(*======================================================================================================================================*)
(*FB_TasterBusSimple:	Einfache RS485 Kommunikation für Haus-bus.de Komponenten zum testen 	
						Achtung: Bei dem 6 Fach Taster ist zu Beachten, dass es nur 4 Externe EA/s gibt also 4 LEDs und 4 Taster *)
(*
Date          	| Version    	| created under        	| Author          	| Remark *)
(*====================================================================================================================================================*)
(*29/04/2025   	| 1.00      		| TC3		  		| N.Kersting       | first release *)
(*02/05/2025   	| 1.01      		| TC3		  		| N.Kersting       | Events für die Buttons werden erfolgreich verarbeitet *)
(*02/05/2025   	| 1.02      		| TC3		  		| N.Kersting       | Events für Temp, Helligkeit, Fuehctigkeit erfolgreich Implementier *)
(*02/05/2025   	| 1.03      		| TC3		  		| N.Kersting       | Set Schrittkette für Reset und LED Helligkeit erfolgreich Implementier*)
(*02/05/2025   	| 1.04      		| TC3		  		| N.Kersting       | In und Out Strukturen Implementiert und Startup nach Reset *)
(*02/05/2025   	| 1.05      		| TC3		  		| N.Kersting       | Pingabgfrage*)
(*02/05/2025   	| 1.06      		| TC3		  		| N.Kersting       | Reset Startup Implementiert*)
(*03/05/2025   	| 1.07      		| TC3		  		| N.Kersting       | Ping wird nun bei PLC Reset auch gestaret und Execute wird richtig verwendet*)
(*04/05/2025   	| 1.08      		| TC3		  		| N.Kersting       | Hintergrundbeleuchtung und Zähler für die Tatser Implementiert *)
(*04/05/2025   	| 1.09      		| TC3		  		| N.Kersting       | Neuen Baustein zum Einheitlichen versenden von Telegrammen Implementiert *)
(*05/05/2025   	| 2.00      		| TC3		  		| N.Kersting       | Komplett neuen Baustein, mit Externer Receive Auswertung und neuem Ping Baustein *)
(*06/05/2025   	| 2.01      		| TC3		  		| N.Kersting       | Externe LEDs Implementiert *)
(*07/05/2025   	| 2.02      		| TC3		  		| N.Kersting       | Im Startup wird nun auf die Device ID geachtet *)
(*08/05/2025   	| 2.03      		| TC3		  		| N.Kersting       | Externe LEDs sind nun Umschaltbar/ LEDs oder normaler Ausgang (Betriefft die Hintergrundbeleuchtung) -> Weniger Busauslastung *)
(*09/05/2025   	| 2.04      		| TC3		  		| N.Kersting       | Ping Versuche Implementiert mit Globalen Parametern *)
(*09/05/2025   	| 2.05      		| TC3		  		| N.Kersting       | Ping für Taster nun Auch automatisch durch Empfang von sämtlichen Telegrammen*)
(*09/05/2025   	| 2.06      		| TC3		  		| N.Kersting       | Bugfix im Startup Angepasst! nur noch Hintergrundbeleuchtung setzen! *)
(*10/05/2025   	| 3.00      		| TC3		  		| N.Kersting       | Umstellung auf Externe FiFo Sendebaustein *)
(*13/05/2025   	| 3.01      		| TC3		  		| N.Kersting       | Viele Bugs gefixt, bei Änderung der Ausgängen wird nun eine Anforderung gesetzt  *)
(*13/05/2025   	| 3.02      		| TC3		  		| N.Kersting       | Test für Github *)
(*22/05/2025   	| 3.03      		| TC3		  		| N.Kersting       | Grundaufbau vom BusTaster, jetzt allerdings für ein CYD mit den gleichen Funktionen *)
(*22/05/2025   	| 3.04      		| TC3		  		| N.Kersting       | ServiceFunktionen für CYD Hinzugefügt (Wifi und Webserver Starten)*)
(*23/05/2025   	| 3.05      		| TC3		  		| N.Kersting       | Neue eigene Input Struktur für das CYD Implementiert*)
(*23/05/2025   	| 3.06      		| TC3		  		| N.Kersting       | Auto - Input Fault Detection implementiert (Wenn Taster zu lange aktiviert bleibt ) *)
(*26/05/2025   	| 3.07      		| TC3		  		| N.Kersting       | Updaten im Com Check Baustein, der Zyklische Ping vom CYD wird nun erkannt ) *)
(*28/05/2025   	| 3.08      		| TC3		  		| N.Kersting       | Neuen Einfachen Ping Baustein, welcher nicht sendet, nur auswertet implementiert *)
(*====================================================================================================================================================*)
FUNCTION_BLOCK fb_CYDBus6F
VAR_INPUT
	I_FifoID			:INT;
	I_bPingStart		:BOOL;						(* Ping Done vom Vorheriegen*)
	I_stInput			:ST_BusCYD6F_Input;
	I_StringReceived	:STRING(255);
END_VAR
VAR_OUTPUT
	Q_sFiFoSend			:STRING(255);
   	Q_stOutput			:ST_BusTaster6F_Output;
	Q_stCnt				:ST_BusTaster6F_Cnt;
END_VAR
VAR
(*----------------------------------------------*)
(* Interne Parameter*)
(*----------------------------------------------*)		
	bSetExecute			:BOOL := TRUE;				(* Aktiviert die Schrittketten, welche Telegramme versenden *)
	bCheckPing			:BOOL := TRUE;				(* Ping Checken Schrittkette Aktivieren *)
	sStartZeichen		:BYTE := 16#FD;				(* Startzeichen Präfix *)
	sEndZeichen			:BYTE := 16#FE;				(* Endzeichen Suffix *)
	iAnzResetSend		:INT := 2;					(* Anzahl der Sendeversuche bei Reset *)
	tPingTimer			:TIME:= T#5S;				(* Zeit, bis wiederholend der Ping versendet wird *)
	tReceiveTimeout		:TIME:= T#2S;				(* Zeit, bis die Event Schrittkette für das Empfangen Automatisch neu Startet*)
	tStartupLEDOn		:TIME:= T#4S;				(* Zeit, wie Lange die LEDS beim Startup kurz eingeschaltet werden *)
	tResetTimeout		:TIME:= T#25S;				(* Zeit, bis bei einem Reset es zu einem Fehler kommt, wenn kein Ping empfangen wird *)
	tResetReboot		:TIME:= T#10S;				(* Zeit, die nach einem Reset Abgewaretet wird damit das Gerät neustarten kann*)
	tResetStartup		:TIME:= T#5S;				(* Zeit, die nach einem Reset Abgewaretet wird bis ein Startup ausgeführt wird nach dem erhalt des Pings vom Gerät*)
	tStartupAfterReset	:TIME := T#5S;				(* Zeit, wann das Startup Zurückgesetzt wird, wenn der Ping verloren wird *)
	bInputFaultDetect	:BOOL := TRUE;				(* Prüft die Eingänge ob sie zu lange geschaltet wurden und führt ein reset des eingangs aus *)
	tInputFaultDetect	:TIME := T#10S;				(* Prüft die Eingänge ob sie zu lange geschaltet wurden und führt ein reset des eingangs aus *)
(*----------------------------------------------*)
(*	Service Funktionen Aktivieren *)
(*----------------------------------------------*)	
	bWebServer			:BOOL := FALSE;				(* zuerst funktion auswählen (bWebserver/ bWifi, bService) und dann mit bStartServiceMode ausführen *)
	bWifi				:BOOL := FALSE;				(* zuerst funktion auswählen (bWebserver/ bWifi, bService) und dann mit bStartServiceMode ausführen *)
	bService			:BOOL := FALSE;				(* zuerst funktion auswählen (bWebserver/ bWifi, bService) und dann mit bStartServiceMode ausführen *)
	(*	*)
	bStartServiceMode	:BOOL := FALSE;				(* zuerst ServiceMode Aktivieren und dann mit bStartServiceMode ausführen *)
	
	(* Speichern der zustände *)
	bMemWebServer		:BOOL;
	bMemWifi			:BOOL;
	bMemService			:BOOL;
	
(*----------------------------------------------*)
(* Strings *)
(*----------------------------------------------*)			
	sSendString			:STRING(255);
	sFiFoSend			:STRING(255);
	sReceived			:STRING(255);
	sLastSendString		:STRING(255);
	sStateReset			:STRING;
(*----------------------------------------------*)
(* Funktionsbausteine *)
(*----------------------------------------------*)
	fbBusTasterEvent	:ARRAY[1..6] OF fb_BusTasterEvent;		(* Interne 6 Taster Abfragen *)
	fbBusTasterEventExt	:ARRAY[1..6] OF fb_BusTasterEvent;		(* Externe 6 Eingänge Abfragen *)
	fbBusTempEvent		:fb_BusTempEvent;
	fbBusBrsEvent		:fb_BusBrsEvent;
	fbBusRhdEvent		:fb_BusRhdEvent;
	fbStringConvTB6F	:fb_StringConvTB6F;
	fbStringConvWeb		:fb_StringConvCYDWeb;
	fbStringConvWifi	:fb_StringConvCYDWifi;
	fbStringConvService	:fb_StringConvCYDService;
	fbPing				:fb_RS485Ping;
(*----------------------------------------------*)
(* Indexe *)
(*----------------------------------------------*)	
	iDeviceStartup		:INT :=0;	(* Startup Schrittkette *)
	sDeviceStartup		:STRING;
    iState     			:INT := 0;
	iStepSet			:INT;
	i,h,j,l,e			:INT;
	idxLED				:INT;
	idxBtn				:INT := 1;
	
	iDimmMem			:ARRAY[1..6] OF INT;
	iDimmMemExt			:ARRAY[1..6] OF INT;
	iDimmBGAnf			:INT;
	iDimmAnf			:ARRAY[1..6] OF INT;
	iDimmAnfExt			:ARRAY[1..6] OF INT;
	
	iDimmBgMem			:INT;
	cntChangesDimm		:INT;
	cntChangesDimmExt	:INT;
	icntResetSend		:INT;
	iMaxPingTry			:INT := 5;
(*----------------------------------------------*)
(* Timer/Trigger *)
(*----------------------------------------------*)		
	r_trigStartupAfterReset	:r_trig;
	r_TrigReset				:r_trig;		
	r_TrigCountBtn			:ARRAY[1..6] OF r_trig;
	
	tonStartupAfterReset	:ton;
	tonReceiveTimeout		:ton;
	tonResetTimeout			:ton;
	tonResetDone			:ton;
	tonStepStartup			:ton;
(*----------------------------------------------*)
(* Status *)
(*----------------------------------------------*)			
	bPingOK					:BOOL;
	bErrorEvent				:BOOL;
	bErrorPing				:BOOL;
	bErrorSet				:BOOL;
	bErrorReset				:BOOL;
	bResetBusy				:BOOL;
	bResetDone				:BOOL;
	bResetAutoStart			:BOOL;
	bStartupStart			:BOOL;
	bStartupDone			:BOOL;	
	bMemExt					:BOOL;
	bStartUpCheckPing		:BOOL;
	bActivateSend			:BOOL;
	bReadyToPing			:BOOL;
	bSendeAnforderung		:BOOL;
	bSendeAnforderungExt	:BOOL;
	bSendeAnforderungBG		:BOOL;
	
END_VAR

(*============================================================================================*)
(* Parameter *)
tPingTimer :=		GVL_HausBus_Parameter.cTimePingTimeCYD;
tReceiveTimeout :=	GVL_HausBus_Parameter.cTimeReceiveTimeoutCYD;
bCheckPing :=		GVL_HausBus_Parameter.bUseCYDPing;
iMaxPingTry :=		GVL_HausBus_Parameter.cMaxPingTry;

(* Service *)
bWebServer :=			I_stInput.bWebServer;
bWifi :=				I_stInput.bWifi;
bService :=				I_stInput.bService;
bStartServiceMode :=	I_stInput.bServiceMode;

(*============================================================================================*)
(* Startup Zurücksetzen Reset *)
r_TrigReset(CLK := I_stInput.bReset);

(* Startup Zurücksetzen bei Busverlust *)
tonStartupAfterReset(
	IN := NOT bPingOK
			AND bCheckPing,
	PT:= tStartupAfterReset);

r_trigStartupAfterReset
	(CLK := tonStartupAfterReset.Q);
	
IF NOT I_stInput.bExecute
	OR r_TrigReset.Q
	OR r_trigStartupAfterReset.Q
THEN
	iDeviceStartup := 0;
ELSIF
	bStartServiceMode
THEN	
	iDeviceStartup := 5;
END_IF

(*============================================================================================*)
(* Ping Dauerhaft Senden*)
ac02_Ping();
	
(*============================================================================================*)
(* Startup Schrittkette *)
CASE iDeviceStartup OF
(*============================================================================================*)
0: 	sDeviceStartup := 'INIT';
	bResetDone := FALSE;
	bStartupDone := FALSE;
	bStartupStart := FALSE;
	bResetAutoStart := FALSE;
	bStartUpCheckPing := FALSE;
	bActivateSend := FALSE;
	bReadyToPing := TRUE;
	bMemWebServer :=FALSE;
	bMemWifi :=	FALSE;
	bMemService	:= FALSE;
	
	sFiFoSend := ''; 
	iStepSet := 0;
	
	IF 	I_stInput.bExecute
	THEN
		iDeviceStartup := iDeviceStartup+1;
	END_IF
(*============================================================================================*)
1: 	sDeviceStartup := 'Device ID Prüfen';
	
	IF  I_stInput.diID <> 0
	THEN
		iDeviceStartup := iDeviceStartup+1;
	ELSE
		sDeviceStartup := 'ERROR- Device ID Prüfen';
	END_IF
(*============================================================================================*)
2: 	sDeviceStartup := 'Verbindung Prüfen';
	bActivateSend := TRUE;	(* Senden Aktivieren *)
	iDeviceStartup := iDeviceStartup+1;
	
	(*
	sDeviceStartup := CONCAT(sDeviceStartup,fbRS485ComCheck.Q_sState);
	
	IF fbRS485ComCheck.Q_bComOk
		OR NOT bCheckPing
	THEN
	END_IF*)

(*============================================================================================*)
3: 	sDeviceStartup := 'Reset Ausführen';	
	bActivateSend := TRUE;	(* Senden Aktivieren *)
	
	(*	RESET Device *)
	ac01_SetReset();
	bResetAutoStart := TRUE;
	
	sDeviceStartup :=	CONCAT(sDeviceStartup,sStateReset);
	
	IF bResetDone
	THEN
		iStepSet := 0;
		iDeviceStartup := iDeviceStartup+1;
	END_IF

(*============================================================================================*)
4: 	sDeviceStartup := 'Startup Ausführen';
		
	(* LED Setzen *)
	ac01_SetLED();
	
	bStartupStart := TRUE;
	
	IF bStartupDone 
	THEN
		bStartupStart := FALSE;
		iDeviceStartup := 999;
	END_IF

(*============================================================================================*)
5:	sDeviceStartup := 'Service Funktionen Steuern';
	ac01_SetService();

	IF NOT bStartServiceMode 
	THEN
		iStepSet := 0;
		iDeviceStartup := 0;
	END_IF
	
(*============================================================================================*)
999: 
	(*bReadyToPing := NOT fbRS485SendCmd.Q_bBusy;*)
	
	(* LED Setzen *)
	ac01_SetLED();
	
	(* Events Auslesen *)
	ac00_Event();
	
	(* Zähler *)
	ac10_Counter();
	
	sDeviceStartup := 'Startup Ausgeführt- Gerät im OP';
	
END_CASE

(*============================================================================================*)
(* Sendebaustein *)
IF bActivateSend
THEN
	Q_sFiFoSend :=	sFiFoSend;
END_IF

(*============================================================================================*)	
(* Zähler *)
ac10_Counter();
	
(*============================================================================================*)
(* Outputs *)
Q_stOutput.bCOM :=		bPingOK;

Q_stOutput.bError := 	bErrorEvent
						OR bErrorPing
						OR bErrorSet
						OR (NOT bPingOK
						AND bCheckPing);
						
Q_stOutput.bStartupDone	:=	bStartupDone;

Q_stOutput.sState :=	CONCAT(I_stInput.sName,'| ');
Q_stOutput.sState :=	CONCAT(Q_stOutput.sState, sDeviceStartup);

ACTION ac00_Event:
(*============================================================================================*)
(*	EVENT Schrittkette *)
(*============================================================================================*)
sReceived := I_StringReceived;
	
FOR i := 1 TO 6 BY 1 DO 
	fbBusTasterEvent[i](
		I_bFaultDetection	:=	bInputFaultDetect,
		I_tFaultDetectTime	:=	tInputFaultDetect,
		I_sID:= 				DINT_TO_STRING(I_stInput.diID), 
		I_sInstID:= 			INT_TO_STRING(i+16), 
		I_sReceivedString:= 	sReceived, 
		Q_bOut=> 				Q_stOutput.bButtons[i]);
	
	fbBusTasterEventExt[i](
		I_sID:= 				DINT_TO_STRING(I_stInput.diID), 
		I_sInstID:= 			INT_TO_STRING(i+32), 
		I_sReceivedString:= 	sReceived, 
		Q_bOut=> 				Q_stOutput.bButtonsExt[i]);
		
	fbBusTempEvent(
		I_sID:= 				DINT_TO_STRING(I_stInput.diID), 
		I_sInstID:= 			'1', 
		I_sReceivedString:= 	sReceived, 
		Q_lrTemp=> 				Q_stOutput.lrTemp);
		
	fbBusBrsEvent(
		I_sID:= 				DINT_TO_STRING(I_stInput.diID), 
		I_sInstID:= 			'1', 
		I_sReceivedString:= 	sReceived, 
		Q_lrBrs=> 				Q_stOutput.lrBrs);
		
	fbBusRhdEvent(
		I_sID:= 				DINT_TO_STRING(I_stInput.diID), 
		I_sInstID:= 			'1', 
		I_sReceivedString:= 	sReceived, 
		Q_lrRhd=> 				Q_stOutput.lrRhd);
END_FOR
END_ACTION

ACTION ac01_SetLED:
(*============================================================================================*)
(*	LED Helligkeit Setzen/ Startup Schrittkette *)
(*============================================================================================*)

(* Einfaches Setzen der LED Helligkeiten (0-100 Prozent *)
(* Neu, es werden alle LEDs zu einem String zusammengefügt und Gleichzeitig gesetzt *)
tonStepStartup(
	PT:= tStartupLEDOn);
	
cntchangesDimm := 0;
cntChangesDimmExt :=0;
	
FOR l := 1 TO 6 BY 1 DO
	IF iDimmMem[l] <> I_stInput.iLED[l]
	THEN
		cntChangesDimm := cntChangesDimm +1;
	END_IF

	IF  iDimmMemExt[l]<> I_stInput.iLEDExt[l]
	THEN
		cntChangesDimmExt := cntChangesDimmExt +1;
	END_IF
END_FOR

CASE iStepSet OF
(*============================================================================================*)
0:	(* INIT und warten auf Change *)				
	tonStepStartup.IN := FALSE;
	sFiFoSend := ''; 
	
	(* Änderungs- Anforderungen Prüfen*)
	FOR e := 1 TO 6 BY 1 DO
		IF cntChangesDimm<>0
		THEN
			(* Helligkeitanforderung Interne LEDs speichern *)
			bSendeAnforderung := TRUE;
			iDimmAnf[e] 	:= I_stInput.iLED[e];
		END_IF
		
		IF cntChangesDimmExt <> 0
		THEN
			(* Helligkeitanforderung Externe LEDs speichern *)
			bSendeAnforderungExt := TRUE;
			iDimmAnfExt[e] 	:= I_stInput.iLEDExt[e];
		END_IF
		
		IF I_stInput.iLEDBg <>iDimmBgMem
		THEN
			(* Helligkeitsanforderung Hintergrundbeleuchtung *)
			bSendeAnforderungBG := TRUE;
			iDimmBGAnf		:= I_stInput.iLEDBg;
		END_IF
	END_FOR
	
	(* Reagieren auf Anforderungen *)
	IF ((bSendeAnforderung
		OR bSendeAnforderungExt
		OR bSendeAnforderungBG)
		AND bSetExecute)
		AND NOT bStartupStart
	THEN
		(* Helligkeitsvorgaben speichern in Mem Arrays *)
		FOR h := 1 TO 6 BY 1 DO
			iDimmMem[h] := I_stInput.iLED[h];
			iDimmMemExt[h] := I_stInput.iLEDExt[h];
			iDimmBgMem := I_stInput.iLEDBg;
		END_FOR
		
		iStepSet := 10;
	ELSIF
		bStartupStart
	THEN
		iStepSet := 100;	(* Startup *)
	END_IF
	
(*============================================================================================*)
10:	(* Prüfen welche Anforderung ausgeführt werden soll *)	
	IF	bSendeAnforderungBG
		AND NOT bSendeAnforderung
		AND NOT bSendeAnforderungExt 
	THEN
		iStepSet := 22;(* Direkt nur die Hintergrund Helligkeit setzen *)
	ELSE
		(* Nur Interne LEDs Schreiben *)
		IF bSendeAnforderung
			AND NOT bSendeAnforderungExt
			AND NOT bSendeAnforderungBG
		THEN
			fbStringConvTB6F(
				I_bSetBackground :=	FALSE,
				I_bReset :=			FALSE,
				I_bExtLED :=		FALSE,
				I_bHasExtLED :=		I_stInput.bExtOutLED,
				I_diID:= 			I_stInput.diID, 
				I_iLED:= 			iDimmAnf, 
				I_iLEDExt:=			iDimmAnfExt,
				I_iLEDBg:= 			iDimmBGAnf,		 
				I_sStartZeichen:= 	sStartZeichen, 
				I_sEndZeichen:= 	sEndZeichen, 
				Q_sConvString=> 	sSendString);
				
			(* Senden an FiFo*)
			IF GVL_RS485FiFoSend.bSendDoneFiFo[I_FifoID]
			THEN
				sFiFoSend :=	sSendString;
			END_IF
			IF NOT GVL_RS485FiFoSend.bSendDoneFiFo[I_FifoID]
			THEN
				bSendeAnforderung := FALSE;
				sLastSendString :=	sFiFoSend;
				iStepSet := 20;
			END_IF
		ELSIF
			(* Nur Externe LEDs Schreiben *)	
			bSendeAnforderungExt
			AND NOT bSendeAnforderung
			AND NOT bSendeAnforderungBG
		THEN
			fbStringConvTB6F(
				I_bSetBackground :=	FALSE,
				I_bReset :=			FALSE,
				I_bExtLED :=		TRUE,
				I_bHasExtLED :=		I_stInput.bExtOutLED,
				I_diID:= 			I_stInput.diID, 
				I_iLED:= 			iDimmAnf, 
				I_iLEDExt:=			iDimmAnfExt,
				I_iLEDBg:= 			iDimmBGAnf,				 
				I_sStartZeichen:= 	sStartZeichen, 
				I_sEndZeichen:= 	sEndZeichen, 
				Q_sConvString=> 	sSendString);
			
			(* Senden an FiFo*)
			IF GVL_RS485FiFoSend.bSendDoneFiFo[I_FifoID]
			THEN
				sFiFoSend :=	sSendString;
			END_IF
			IF NOT GVL_RS485FiFoSend.bSendDoneFiFo[I_FifoID]
			THEN
				bSendeAnforderungExt := FALSE;
				sLastSendString :=	sFiFoSend;
				iStepSet := 20;
			END_IF
		ELSE
			(* Externe und Interne LEDs Schreiben *)
			bMemExt := TRUE; (* Speichern, damit anschließend noch die Externen LEDs gesetzt werden *)
			
			fbStringConvTB6F(
				I_bSetBackground :=	FALSE,
				I_bReset :=			FALSE,
				I_bExtLED :=		FALSE,
				I_bHasExtLED :=		I_stInput.bExtOutLED,
				I_diID:= 			I_stInput.diID, 
				I_iLED:= 			iDimmAnf, 
				I_iLEDExt:=			iDimmAnfExt,
				I_iLEDBg:= 			iDimmBGAnf,			 
				I_sStartZeichen:= 	sStartZeichen, 
				I_sEndZeichen:= 	sEndZeichen, 
				Q_sConvString=> 	sSendString);
			
			(* Senden an FiFo*)
			IF GVL_RS485FiFoSend.bSendDoneFiFo[I_FifoID]
			THEN
				sFiFoSend :=	sSendString;
			END_IF
			IF NOT GVL_RS485FiFoSend.bSendDoneFiFo[I_FifoID]
			THEN
				bSendeAnforderung := FALSE;
				bSendeAnforderungExt := FALSE;
				sLastSendString :=	sFiFoSend;
				iStepSet := 20;
			END_IF
		END_IF
	END_IF
(*============================================================================================*)	
20:	(* Warten bis nicht Busy *)	
	
	IF GVL_RS485FiFoSend.bSendDoneFiFo[I_FifoID]
	THEN
		sFiFoSend := ''; 
		IF NOT bMemExt
		THEN
			IF bSendeAnforderungBG
			THEN
				iStepSet := 22;
			ELSE
				iStepSet := 0;
			END_IF
		ELSE
			iStepSet :=	21;
		END_IF
	END_IF
	
(*============================================================================================*)	
21:	(* Externe LEDs Senden *)	
	bMemExt := FALSE;
	bSendeAnforderungExt := FALSE;
	
	fbStringConvTB6F(
		I_bSetBackground :=	FALSE,
		I_bReset :=			FALSE,
		I_bExtLED :=		TRUE,
		I_bHasExtLED :=		I_stInput.bExtOutLED,
		I_diID:= 			I_stInput.diID, 
		I_iLED:= 			iDimmAnf, 
		I_iLEDExt:=			iDimmAnfExt,
		I_iLEDBg:= 			iDimmBGAnf,				 
		I_sStartZeichen:= 	sStartZeichen, 
		I_sEndZeichen:= 	sEndZeichen, 
		Q_sConvString=> 	sSendString);
		
	(* Senden an FiFo*)
	IF GVL_RS485FiFoSend.bSendDoneFiFo[I_FifoID]
	THEN
		sFiFoSend :=	sSendString;
	END_IF
	IF NOT GVL_RS485FiFoSend.bSendDoneFiFo[I_FifoID]
	THEN
		sLastSendString :=	sFiFoSend;
		iStepSet := 20;
	END_IF
	
(*============================================================================================*)	
22:	(* Hintergrundbeleuchtung senden *)		
	bSendeAnforderungBG := FALSE;
	
	fbStringConvTB6F(
		I_bSetBackground :=	TRUE,
		I_bReset :=			FALSE,
		I_bExtLED :=		FALSE,
		I_bHasExtLED :=		I_stInput.bExtOutLED,
		I_diID:= 			I_stInput.diID, 
		I_iLED:= 			iDimmAnf, 
		I_iLEDExt:=			iDimmAnfExt,
		I_iLEDBg:= 			iDimmBGAnf,			 
		I_sStartZeichen:= 	sStartZeichen, 
		I_sEndZeichen:= 	sEndZeichen, 
		Q_sConvString=> 	sSendString);
		
	(* Senden an FiFo*)
	IF GVL_RS485FiFoSend.bSendDoneFiFo[I_FifoID]
	THEN
		sFiFoSend :=	sSendString;
	END_IF
	IF NOT GVL_RS485FiFoSend.bSendDoneFiFo[I_FifoID]
	THEN
		sLastSendString :=	sFiFoSend;
		iStepSet := 20;
	END_IF

(*============================================================================================*)	
(* Startup LEDS einmal Einschalten *)
100:	tonStepStartup.IN := TRUE;
	
	IF tonStepStartup.Q
	THEN
		iStepSet := 110;
	END_IF
	
(*============================================================================================*)
110:	(* String senden *)	
	tonStepStartup.IN := FALSE;
	
	fbStringConvTB6F(
		I_bSetBackground :=	TRUE,
		I_bExtLED :=		FALSE,
		I_bReset :=			FALSE,
		I_bHasExtLED :=		I_stInput.bExtOutLED,
		I_diID:= 			I_stInput.diID, 
		I_iLEDBg:= 			5,		 
		I_sStartZeichen:= 	sStartZeichen, 
		I_sEndZeichen:= 	sEndZeichen, 
		Q_sConvString=> 	sSendString);
			
	(* Senden an FiFo*)
	IF GVL_RS485FiFoSend.bSendDoneFiFo[I_FifoID]
	THEN
		sFiFoSend :=	sSendString;
	END_IF
	IF NOT GVL_RS485FiFoSend.bSendDoneFiFo[I_FifoID]
	THEN
		
		iStepSet := 111;
	END_IF
	
(*============================================================================================*)	
111:(* Warten bis nicht Busy *)	
	IF GVL_RS485FiFoSend.bSendDoneFiFo[I_FifoID]
	THEN
		sFiFoSend := ''; 
		tonStepStartup.IN := TRUE;
		
		IF tonStepStartup.Q
		THEN
			tonStepStartup.IN := FALSE;
			iStepSet := 120;
		END_IF
	END_IF
	
(*============================================================================================*)
120:	(* String senden *)	
	fbStringConvTB6F(
		I_bSetBackground :=	TRUE,
		I_bExtLED :=		FALSE,
		I_bReset :=			FALSE,
		I_bHasExtLED :=		I_stInput.bExtOutLED,
		I_diID:= 			I_stInput.diID, 
		I_iLEDBg:= 			100,		 
		I_sStartZeichen:= 	sStartZeichen, 
		I_sEndZeichen:= 	sEndZeichen, 
		Q_sConvString=> 	sSendString);
			
	(* Senden an FiFo*)
	IF GVL_RS485FiFoSend.bSendDoneFiFo[I_FifoID]
	THEN
		sFiFoSend :=	sSendString;
	END_IF
	IF NOT GVL_RS485FiFoSend.bSendDoneFiFo[I_FifoID]
	THEN
		iStepSet := 130;
	END_IF
	
(*============================================================================================*)	
130:(* Warten bis nicht Busy *)	
	IF GVL_RS485FiFoSend.bSendDoneFiFo[I_FifoID]
	THEN
		sFiFoSend := ''; 
			
		tonStepStartup.IN := TRUE;
	
		IF tonStepStartup.Q
		THEN
			bStartupDone := TRUE;
			tonStepStartup.IN := FALSE;
			bStartupStart := FALSE;
			iStepSet := 10;	(* Anschließend noch einmal die Eingangs Helligkeit setzen *)
		END_IF
	END_IF	

END_CASE

(*bErrorSet := fbRS485SendCmd.Q_bError;*)
END_ACTION

ACTION ac01_SetReset:
(*============================================================================================*)
(*	RESET Schrittkette *)
(*============================================================================================*)
tonResetTimeout(
	PT := tResetTimeout);

tonResetDone();

(* Einfaches Setzen der LED Helligkeiten (0-100 Prozent *)
CASE iStepSet OF
(*============================================================================================*)
0:	sStateReset := 'INIT';
	
	IF (bSetExecute
		AND (I_stInput.bReset
		OR bResetAutoStart))
	THEN
		sFiFoSend := ''; 
		bStartupDone := FALSE;
		bResetDone := FALSE;
		tonResetTimeout.IN := FALSE;
		tonResetDone.IN := FALSE;
		icntResetSend := 0;
		
		(* Ausgänge alle auf 0 setzen *)
		FOR h := 1 TO 6 BY 1 DO
			fbBusTasterEvent[i](
				I_sReceivedString :='');
				
			fbBusTasterEventExt[i](
				I_sReceivedString :='');	
				
			iDimmMem[h] := 0;
			Q_stOutput.bButtons[h] := FALSE;
			Q_stOutput.lrTemp := 0;
			Q_stOutput.lrBrs := 0;
			Q_stOutput.lrRhd := 0;
		END_FOR
		
		fbBusTempEvent(
			I_sReceivedString :='',	
			I_bReset := TRUE);
			
		fbBusBrsEvent(
			I_sReceivedString :='',	
			I_bReset := TRUE);
			
		fbBusRhdEvent(
			I_sReceivedString :='',	
			I_bReset := TRUE);
		
		bPingOK := FALSE;
		
		iStepSet := iStepSet +1;
	END_IF

(*============================================================================================*)	
1:	sStateReset := 'Sende Reset Befehl';
	bResetBusy := TRUE;
	bErrorReset := FALSE;
	
	fbStringConvTB6F(
		I_bReset :=			TRUE,
		I_diID:= 			I_stInput.diID, 		 
		I_sStartZeichen:= 	sStartZeichen, 
		I_sEndZeichen:= 	sEndZeichen, 
		Q_sConvString=> 	sSendString);

	(* Senden an FiFo*)
	IF GVL_RS485FiFoSend.bSendDoneFiFo[I_FifoID]
	THEN
		sFiFoSend :=	sSendString;
	END_IF
	IF NOT GVL_RS485FiFoSend.bSendDoneFiFo[I_FifoID]
	THEN
		iStepSet := iStepSet+1;
	END_IF

(*============================================================================================*)
2:	sStateReset := 'Sende Reset Befehl';

	IF GVL_RS485FiFoSend.bSendDoneFiFo[I_FifoID]
	THEN
		sFiFoSend := ''; 
		fbStringConvTB6F(
			I_bReset :=			FALSE);
		iStepSet := 3;
				
	END_IF
	
(*============================================================================================*)	
3:	sStateReset := 'Reset durchgeführt, Warte auf Ping';
	tonResetDone.IN := TRUE;
	tonResetDone.PT := tResetReboot;
	
	fbBusTempEvent(I_bReset := FALSE);
	fbBusBrsEvent(I_bReset := FALSE);
	fbBusRhdEvent(I_bReset := FALSE);
	
	iState := 0;
	
	IF tonResetDone.Q
	THEN
		tonResetDone.IN := FALSE;
		iStepSet := 4;
	END_IF
	
(*============================================================================================*)	
4:	sStateReset := 'Warte auf Ping vom Gerät';	
	tonResetTimeout.IN := TRUE;
	bStartUpCheckPing := TRUE;
	
	IF bPingOK 
	(*	OR NOT bCheckPing*)
	THEN
		bErrorReset := FALSE;
		tonResetTimeout.IN := FALSE;
		iStepSet := 5;
	ELSIF
		tonResetTimeout.Q
	THEN
		sStateReset := 'Ping Timeout, keine Kommunikation';
		bErrorReset := TRUE;

		IF I_stInput.bReset
		THEN
			bResetBusy := FALSE;
			iStepSet := 0;
		END_IF
	END_IF

(*============================================================================================*)
5:	sStateReset := 'Startup Aktiv';
	
	tonResetDone.IN := NOT I_stInput.bReset;
	tonResetDone.PT := tResetStartup;
	sFiFoSend := ''; 
	
	IF tonResetDone.Q
	THEN
		fbStringConvTB6F(
			I_bReset :=			FALSE);
			
		sStateReset := 'Ping erhalten, Reset Erfolgreich';
		bResetAutoStart := FALSE;
		bResetDone := TRUE;
		bResetBusy := FALSE;
		iState := 0;
		iStepSet := 0;
	END_IF
END_CASE
END_ACTION

ACTION ac01_SetService:
(*============================================================================================*)
(*	RESET Schrittkette *)
(*============================================================================================*)
tonResetTimeout(
	PT := tResetTimeout);

tonResetDone();

(* Einfaches Setzen der LED Helligkeiten (0-100 Prozent *)
CASE iStepSet OF
(*============================================================================================*)
0:	sStateReset := 'INIT';
	
	IF bSetExecute
		AND (bMemWebServer <> bWebServer
		OR bMemWifi <> bWifi
		OR bMemService <> bService )
	THEN
		bMemWebServer :=	bWebServer;
		bMemWifi :=			bWifi;
		bMemService	:=		bService;
		
		sFiFoSend := ''; 
		tonResetTimeout.IN := FALSE;
		tonResetDone.IN := FALSE;
		icntResetSend := 0;
		
		iStepSet := iStepSet +1;
	END_IF

(*============================================================================================*)	
1:	sStateReset := 'Sende Webserver Befehl';
	fbStringConvWeb(
		I_diID:= 			I_stInput.diID,
		I_bWebOn:= 			bWebServer, 
		I_sStartZeichen:= 	sStartZeichen, 
		I_sEndZeichen:= 	sEndZeichen, 
		Q_sConvString=> 	sSendString);
	
	(* Senden an FiFo*)
	IF GVL_RS485FiFoSend.bSendDoneFiFo[I_FifoID]
	THEN
		sFiFoSend :=	sSendString;
	END_IF
	IF NOT GVL_RS485FiFoSend.bSendDoneFiFo[I_FifoID]
	THEN
		iStepSet := iStepSet+1;
	END_IF

(*============================================================================================*)
2:	sStateReset := 'Sende Webserver Befehl';

	IF GVL_RS485FiFoSend.bSendDoneFiFo[I_FifoID]
	THEN
		sFiFoSend := ''; 
		iStepSet := 3;
	END_IF
	
(*============================================================================================*)	
3:	sStateReset := 'Sende Wifi Befehl';
	
	fbStringConvWifi(
		I_diID:= 			I_stInput.diID,
		I_bWifiOn:= 		bWifi, 
		I_sStartZeichen:= 	sStartZeichen, 
		I_sEndZeichen:= 	sEndZeichen, 
		Q_sConvString=> 	sSendString);
	
	(* Senden an FiFo*)
	IF GVL_RS485FiFoSend.bSendDoneFiFo[I_FifoID]
	THEN
		sFiFoSend :=	sSendString;
	END_IF
	IF NOT GVL_RS485FiFoSend.bSendDoneFiFo[I_FifoID]
	THEN
		iStepSet := iStepSet+1;
	END_IF
	
(*============================================================================================*)	
4:	sStateReset := 'Sende Wifi Befehl';

	IF GVL_RS485FiFoSend.bSendDoneFiFo[I_FifoID]
	THEN
		sFiFoSend := ''; 
		iStepSet := 5;
	END_IF
(*============================================================================================*)	
5:	sStateReset := 'Sende Service Befehl';
	
	fbStringConvService(
		I_diID:= 			I_stInput.diID,
		I_bServiceOn:= 		bService, 
		I_sStartZeichen:= 	sStartZeichen, 
		I_sEndZeichen:= 	sEndZeichen, 
		Q_sConvString=> 	sSendString);
	
	(* Senden an FiFo*)
	IF GVL_RS485FiFoSend.bSendDoneFiFo[I_FifoID]
	THEN
		sFiFoSend :=	sSendString;
	END_IF
	IF NOT GVL_RS485FiFoSend.bSendDoneFiFo[I_FifoID]
	THEN
		iStepSet := iStepSet+1;
	END_IF
	
(*============================================================================================*)	
6:	sStateReset := 'Sende Service Befehl';

	IF GVL_RS485FiFoSend.bSendDoneFiFo[I_FifoID]
	THEN
		sFiFoSend := ''; 
		iStepSet := 7;
	END_IF
	
(*============================================================================================*)
7:	sStateReset := 'Fertig';
	
	IF bMemWebServer <> bWebServer
		OR bMemWifi <> bWifi
		OR bMemService <> bService 
	THEN
		iStepSet := 0;
	END_IF
	
END_CASE
END_ACTION

ACTION ac02_Ping:
(*============================================================================================*)
(* 	Ping Bautsein, Checkt ob die Kommunikation vorhanden ist *)
(*============================================================================================*)
fbPing(
	I_bExecute:= 			bStartUpCheckPing, 
	I_bAutoPing:= 			bCheckPing, 
	I_bAutoReset:= 			bCheckPing, 
	I_bReset:= 				r_TrigReset.Q
							OR NOT bStartUpCheckPing, 
	I_tPingTimeout:= 		tPingTimer, 
	I_diID:= 				I_stInput.diID, 
	I_sStartZeichen:= 		sStartZeichen, 
	I_sEndZeichen:= 		sEndZeichen, 
	I_StringReceived:= 		I_StringReceived, 
	Q_sState=> , 
	Q_bComOk=> 				bPingOK, 
	Q_bTimeout=> 			bErrorPing);
END_ACTION

ACTION ac10_Counter:
(*============================================================================================*)
(* 	Zähler *)
(*============================================================================================*)
FOR j := 1 TO 6 BY 1 DO 
	r_TrigCountBtn[j](
		CLK := Q_stOutput.bButtons[j]);
		
	IF r_TrigCountBtn[j].Q
	THEN
		Q_stCnt.dwCntButtons[j] := Q_stCnt.dwCntButtons[j]+1;
	END_IF
	
END_FOR
END_ACTION

ACTION ac99_Doku:
(*======================================================================================================================================*)
(*	DOKU	*)
(*======================================================================================================================================*)
(* Wichtiger Hinweis:
		-Bei dem 6 Fach Taster ist zu Beachten, dass es nur 4 Externe EA/s gibt also 4 LEDs und 4 Taster, 
		da der ESP 32 Nur 10Es und 10As besitzt.
		- Die 4 Zusätzlichen Ausgänge werden von der Hintergrundbeleuchtung Ausgeschlossen und müssen über den Befehl: SET_MBR einzeln 
			gesetzt werden! *)	
	
(* Verdrahtung:		
	Verdrahtung füR: KL6041
        +-------+
        |       |
        | TxD+ ----+
        |         |----> RS485 A (zum Bus)
        | RxD+ ----+
        |         |
        | TxD− ----+
        |         |----> RS485 B (zum Bus)
        | RxD− ----+
        +-------+	*)
		
(*======================================================================================================================================*)
(* Telegrammbeschreibung *)

(*	Die XML Dateien der verschiedenen Module sind grundsätzlich immer gleich aufgebaut. 
	Je Instanz der verschiedenen Sensoren und Aktoren werden die zu sendenden Befehle bzw. 
	die zu empfangenen Events beschrieben. 
	Alle Telegramme sind ASCII kodiert und sind umgeben mit dem binären Startzeichen 0xFD und dem binären Endezeichen 0xFE.

	Grundaufbauer aller im Folgenden beschriebenen Telegramme:
	
	-Startzeichen immer 0xFD.
	-Punkte dienen als Trennzeichen der verschiedenen Elemente
	-Endezeichen immer 0xFE.
	-Element 1 ist die Geräte-ID, die entsprechend der verwendeten Module angepasst werden muss (hier beispielhaft jeweils 12345)
	-Element 2 ist ein Schlüsselwort für den jeweiligen Funktionstyp (z.b. BTN, LED, DIM, usw)
	-Element 3 ist die InstanzID gemäß XML Templates (also welche Taster oder welcher Dimmer konkret gemeint ist)
	-Element 4 zeigt die jeweilige Aktion zum Funktionstypen (z.b. ON, OFF, STATUS)
	-Anschließend kommen optional diverse Parameter, die mit P1,P2,...P3 bezeichnet werden
	
	Im Folgenden wird nur noch auf die speziellen Telegramdaten eingegangen:
	
	(*------------------------------------------------------------*)
	Taster oder digitaler Eingang (Sensor):
	(*------------------------------------------------------------*)
	Telegram Event:  	
	
	\xFD 12345.BTN.17.STATUS.P1 \xFE
	
		Funktionstyp:		BTN (kurz für Button)
		Instanz-ID:			hier 17 (in XML nachschauen)
		Aktion:				STATUS
		P1:					1, wenn Taste gedrückt bzw. Eingang aktiv
							0, wenn Taste losgelassen bzw. Eingang inaktiv
	
	Telegram Statusabfrage:  	
	
	\xFD 12345.BTN.17.gSTATUS \xFE
	
		Antwort:  			\xFD 12345.BTN.17.rSTATUS.P1 \xFE
		P1:					1, wenn Taste gedrückt bzw. Eingang aktiv
							0, wenn Taste losgelassen bzw. Eingang inaktiv

	(*------------------------------------------------------------*)
	Led (Aktor):
	(*------------------------------------------------------------*)
	Telegram Helligkeit setzen:  	
	
	\xFD 12345.LED.50.ON.P1.P2.P3 \xFE
	
		Funktionstyp:			LED
		Instanz-ID:				hier 50 (in XML nachschauen)
		Aktion:					ON
		P1:						gewünschte Helligkeit 0-100
		P2:						Einschaltdauer in 100stel Sekunden (0 = daueran)
		P3:						Einschaltverzögerung in Sekunden (0 = ohne Verzögerung)
	
	Telegram Mindesthelligkeit:  	
	
	\xFD 12345.LED.50.SET_MBR.P1 \xFE
		
		Aktion:					SET_MBR (Setzt eine Mindesthelligkeit, die auch dann erhalten bleibt, wenn man per OFF ausschaltet)
		P1:						gewünschte Helligkeit 0-100
	
	Telegram Statusabfrage:  	

	\xFD 12345.LED.50.gSTATUS \xFE
	
		Antwort:  				\xFD 12345.LED.50.rSTATUS.P1.P2 \xFE
		P1:						aktuelle Helligkeit 0-100
		P2:						Einschaltdauer in 100stel Sekunden
	
	(*------------------------------------------------------------*)
	Hintergrundbeleuchtung (Aktor):
	(*------------------------------------------------------------*)
	Telegram Minhelligkeit:  
	
	\xFD 12345.LBN.16.SET_MBR.P1 \xFE
	
		Aktion:					SET_MBR ((Setzt eine Mindesthelligkeit, die auch dann erhalten bleibt, wenn man per OFF ausschaltet)
		P1:						gewünschte Helligkeit 0-100
		
	Telegram Statusabfrage:  	

	\xFD 12345.LBN.16.gSTATUS \xFE
	
		Antwort:  				\xFD 12345.LBN.16.rSTATUS.P1 \xFE
		P1:						aktuelle Helligkeit 0-100

	(*------------------------------------------------------------*)
	Temperatursensor (Sensor):
	(*------------------------------------------------------------*)
	Telegram Event:  	
	
	\xFD 12345.TMP.1.STATUS.P1.P2 \xFE
	
		Funktionstyp:			TMP (kurz für Temperatur)
		Instanz-ID:				hier 1 (in XML nachschauen)
		Aktion:					STATUS
		P1:						Temperatur in Grad Vorkommastellen
		P2:						Temperatur in Grad Nachkommastellen
	
	Telegram Statusabfrage:  
	
	\xFD 12345.TMP.1.gSTATUS \xFE
	
		Antwort:  				\xFD 12345.TMP.1.rSTATUS.P1.P2 \xFE
		P1:						Temperatur in Grad Vorkommastellen
		P2:						Temperatur in Grad Nachkommastellen

	(*------------------------------------------------------------*)
	Feuchtesensor (Sensor):
	(*------------------------------------------------------------*)
	Telegram Event:  	

	\xFD 12345.RHD.1.STATUS.P1.P2 \xFE
	
		Funktionstyp:			RHD (kurz für Relative Humidity)
		Instanz-ID:				hier 1 (in XML nachschauen)
		Aktion:					STATUS
		P1:						Relative Luftfeuchtigkeit 0-100 Vorkommastellen
		P2:						Relative Luftfeuchtigkeit 0-100 Nachkommastellen

	Telegram Statusabfrage:  	
	
	\xFD 12345.RHD.1.gSTATUS \xFE
	
	Antwort:  					\xFD 12345.RHD.1.rSTATUS.P1 \xFE
	P1:							Relative Luftfeuchtigkeit 0-100 Vorkommastellen
	P2:							Relative Luftfeuchtigkeit 0-100 Nachkommastellen

	(*------------------------------------------------------------*)
	Helligkeitssensor (Sensor):
	(*------------------------------------------------------------*)
	Telegram Event:  	
	
	\xFD 12345.BRS.23.STATUS.P1.P2 \xFE
	
		Funktionstyp:			BRS (kurz für Brightness Sensor)
		Instanz-ID:				hier 23 (in XML nachschauen)
		Aktion:					STATUS
		P1:						Relative Helligkeit 0-255 Vorkommastellen
		P2:						Relative Helligkeit 0-255 Nachkommastellen
	
	Telegram Statusabfrage:  	
	
	\xFD 12345.BRS.23.gSTATUS \xFE
	
	Antwort:  					\xFD 12345.BRS.23.rSTATUS.P1 \xFE
	P1:							Relative Helligkeit 0-255 Vorkommastellen
	P2:							Relative Helligkeit 0-255 Nachkommastellen

(*======================================================================================================================================*)
(* Alle Telegramme im Überblick *)	

	<?xml version="1.0" encoding="utf-8"?>
	<Comm Title="Haus-Bus ID 12345" Comment="" Baudrate="57600" Databits="8" Parity="1" EndChar="510">
	<CommCmd Title="6-fach Taster 12345 - Hintergrundbeleuchtung" Comment="" CmdOn="\xFD12345.LBN.16.SET_MBR.&lt;v&gt;.0\xFE" CmdOff="\xFD12345.LBN.16.SET_MBR.0\xFE" Unit="" Analog="true" Text="false" Sensor="false" SourceValHigh="100" DestValHigh="100"/>
	<CommCmd Title="6-fach Taster 12345 - Temperatursensor" Comment="" CmdOn="\xFD12345.TMP.1.STATUS.\v\xFE" CmdOff="" Unit="&lt;v.2&gt;" Analog="true" Text="false" Sensor="true" SourceValHigh="100" DestValHigh="100"/>
	<CommCmd Title="6-fach Taster 12345 - Feuchtesensor" Comment="" CmdOn="\xFD12345.RHD.1.STATUS.\v\xFE" CmdOff="" Unit="&lt;v.x&gt;" Analog="true" Text="false" Sensor="true" SourceValHigh="100" DestValHigh="100"/>
	<CommCmd Title="6-fach Taster 12345 - Helligkeitssensor" Comment="" CmdOn="\xFD12345.BRS.1.STATUS.\v\xFE" CmdOff="" Unit="&lt;v.x&gt;" Analog="true" Text="false" Sensor="true" SourceValHigh="100" DestValHigh="100"/>
	<CommCmd Title="6-fach Taster 12345 - Led 1" Comment="" CmdOn="\xFD12345.LED.49.ON.&lt;v&gt;.0\xFE" CmdOff="\xFD12345.LED.49.OFF\xFE" Unit="" Analog="true" Text="false" Sensor="false" SourceValHigh="100" DestValHigh="100"/>
	<CommCmd Title="6-fach Taster 12345 - Led 2" Comment="" CmdOn="\xFD12345.LED.50.ON.&lt;v&gt;.0\xFE" CmdOff="\xFD12345.LED.50.OFF\xFE" Unit="" Analog="true" Text="false" Sensor="false" SourceValHigh="100" DestValHigh="100"/>
	<CommCmd Title="6-fach Taster 12345 - Led 3" Comment="" CmdOn="\xFD12345.LED.51.ON.&lt;v&gt;.0\xFE" CmdOff="\xFD12345.LED.51.OFF\xFE" Unit="" Analog="true" Text="false" Sensor="false" SourceValHigh="100" DestValHigh="100"/>
	<CommCmd Title="6-fach Taster 12345 - Led 4" Comment="" CmdOn="\xFD12345.LED.52.ON.&lt;v&gt;.0\xFE" CmdOff="\xFD12345.LED.52.OFF\xFE" Unit="" Analog="true" Text="false" Sensor="false" SourceValHigh="100" DestValHigh="100"/>
	<CommCmd Title="6-fach Taster 12345 - Led 5" Comment="" CmdOn="\xFD12345.LED.53.ON.&lt;v&gt;.0\xFE" CmdOff="\xFD12345.LED.53.OFF\xFE" Unit="" Analog="true" Text="false" Sensor="false" SourceValHigh="100" DestValHigh="100"/>
	<CommCmd Title="6-fach Taster 12345 - Led 6" Comment="" CmdOn="\xFD12345.LED.54.ON.&lt;v&gt;.0\xFE" CmdOff="\xFD12345.LED.54.OFF\xFE" Unit="" Analog="true" Text="false" Sensor="false" SourceValHigh="100" DestValHigh="100"/>
	<CommCmd Title="6-fach Taster 12345 - Taster 1" Comment="" CmdOn="\xFD12345.BTN.17.STATUS.\v\xFE" CmdOff="" Unit="&lt;v.x&gt;" Analog="true" Text="false" Sensor="true" SourceValHigh="100" DestValHigh="100"/>
	<CommCmd Title="6-fach Taster 12345 - Taster 2" Comment="" CmdOn="\xFD12345.BTN.18.STATUS.\v\xFE" CmdOff="" Unit="&lt;v.x&gt;" Analog="true" Text="false" Sensor="true" SourceValHigh="100" DestValHigh="100"/>
	<CommCmd Title="6-fach Taster 12345 - Taster 3" Comment="" CmdOn="\xFD12345.BTN.19.STATUS.\v\xFE" CmdOff="" Unit="&lt;v.x&gt;" Analog="true" Text="false" Sensor="true" SourceValHigh="100" DestValHigh="100"/>
	<CommCmd Title="6-fach Taster 12345 - Taster 4" Comment="" CmdOn="\xFD12345.BTN.20.STATUS.\v\xFE" CmdOff="" Unit="&lt;v.x&gt;" Analog="true" Text="false" Sensor="true" SourceValHigh="100" DestValHigh="100"/>
	<CommCmd Title="6-fach Taster 12345 - Taster 5" Comment="" CmdOn="\xFD12345.BTN.21.STATUS.\v\xFE" CmdOff="" Unit="&lt;v.x&gt;" Analog="true" Text="false" Sensor="true" SourceValHigh="100" DestValHigh="100"/>
	<CommCmd Title="6-fach Taster 12345 - Taster 6" Comment="" CmdOn="\xFD12345.BTN.22.STATUS.\v\xFE" CmdOff="" Unit="&lt;v.x&gt;" Analog="true" Text="false" Sensor="true" SourceValHigh="100" DestValHigh="100"/>
	<CommCmd Title="6-fach Taster 12345 - Extern Taster 1" Comment="" CmdOn="\xFD12345.BTN.33.STATUS.\v\xFE" CmdOff="" Unit="&lt;v.x&gt;" Analog="true" Text="false" Sensor="true" SourceValHigh="100" DestValHigh="100"/>
	<CommCmd Title="6-fach Taster 12345 - Extern Taster 2" Comment="" CmdOn="\xFD12345.BTN.34.STATUS.\v\xFE" CmdOff="" Unit="&lt;v.x&gt;" Analog="true" Text="false" Sensor="true" SourceValHigh="100" DestValHigh="100"/>
	<CommCmd Title="6-fach Taster 12345 - Extern Taster 3" Comment="" CmdOn="\xFD12345.BTN.35.STATUS.\v\xFE" CmdOff="" Unit="&lt;v.x&gt;" Analog="true" Text="false" Sensor="true" SourceValHigh="100" DestValHigh="100"/>
	<CommCmd Title="6-fach Taster 12345 - Extern Taster 4" Comment="" CmdOn="\xFD12345.BTN.36.STATUS.\v\xFE" CmdOff="" Unit="&lt;v.x&gt;" Analog="true" Text="false" Sensor="true" SourceValHigh="100" DestValHigh="100"/>
	<CommCmd Title="6-fach Taster 12345 - Extern Taster 5" Comment="" CmdOn="\xFD12345.BTN.37.STATUS.\v\xFE" CmdOff="" Unit="&lt;v.x&gt;" Analog="true" Text="false" Sensor="true" SourceValHigh="100" DestValHigh="100"/>
	<CommCmd Title="6-fach Taster 12345 - Extern Taster 6" Comment="" CmdOn="\xFD12345.BTN.38.STATUS.\v\xFE" CmdOff="" Unit="&lt;v.x&gt;" Analog="true" Text="false" Sensor="true" SourceValHigh="100" DestValHigh="100"/>
	<CommCmd Title="6-fach Taster 12345 - Extern Led 1" Comment="" CmdOn="\xFD12345.LED.65.ON.&lt;v&gt;.0\xFE" CmdOff="\xFD12345.LED.65.OFF\xFE" Unit="" Analog="true" Text="false" Sensor="false" SourceValHigh="100" DestValHigh="100"/>
	<CommCmd Title="6-fach Taster 12345 - Extern Led 2" Comment="" CmdOn="\xFD12345.LED.66.ON.&lt;v&gt;.0\xFE" CmdOff="\xFD12345.LED.66.OFF\xFE" Unit="" Analog="true" Text="false" Sensor="false" SourceValHigh="100" DestValHigh="100"/>
	<CommCmd Title="6-fach Taster 12345 - Extern Led 3" Comment="" CmdOn="\xFD12345.LED.67.ON.&lt;v&gt;.0\xFE" CmdOff="\xFD12345.LED.67.OFF\xFE" Unit="" Analog="true" Text="false" Sensor="false" SourceValHigh="100" DestValHigh="100"/>
	<CommCmd Title="6-fach Taster 12345 - Extern Led 4" Comment="" CmdOn="\xFD12345.LED.68.ON.&lt;v&gt;.0\xFE" CmdOff="\xFD12345.LED.68.OFF\xFE" Unit="" Analog="true" Text="false" Sensor="false" SourceValHigh="100" DestValHigh="100"/>
	<CommCmd Title="6-fach Taster 12345 - Extern Led 5" Comment="" CmdOn="\xFD12345.LED.69.ON.&lt;v&gt;.0\xFE" CmdOff="\xFD12345.LED.69.OFF\xFE" Unit="" Analog="true" Text="false" Sensor="false" SourceValHigh="100" DestValHigh="100"/>
	<CommCmd Title="6-fach Taster 12345 - Extern Led 6" Comment="" CmdOn="\xFD12345.LED.70.ON.&lt;v&gt;.0\xFE" CmdOff="\xFD12345.LED.70.OFF\xFE" Unit="" Analog="true" Text="false" Sensor="false" SourceValHigh="100" DestValHigh="100"/>
	<CommCmd Title="6-fach Taster 12345 - RFID Leser" Comment="" CmdOn="\xFD12345.RFD.65.TAG_ID.\v\xFE" CmdOff="" Unit="&lt;v.x&gt;" Analog="false" Text="true" Sensor="true" SourceValHigh="100" DestValHigh="100"/>
	<CommCmd Title="6-fach Taster 12345 - RFID Leser" Comment="" CmdOn="\xFD12345.RFD.66.TAG_ID.\v\xFE" CmdOff="" Unit="&lt;v.x&gt;" Analog="false" Text="true" Sensor="true" SourceValHigh="100" DestValHigh="100"/>
	<CommCmd Title="6-fach Taster 12345 - RFID Leser" Comment="" CmdOn="\xFD12345.RFD.67.TAG_ID.\v\xFE" CmdOff="" Unit="&lt;v.x&gt;" Analog="false" Text="true" Sensor="true" SourceValHigh="100" DestValHigh="100"/>
	<CommCmd Title="6-fach Taster 12345 - RFID Leser" Comment="" CmdOn="\xFD12345.RFD.68.TAG_ID.\v\xFE" CmdOff="" Unit="&lt;v.x&gt;" Analog="false" Text="true" Sensor="true" SourceValHigh="100" DestValHigh="100"/>
	<CommCmd Title="6-fach Taster 12345 - RFID Leser" Comment="" CmdOn="\xFD12345.RFD.69.TAG_ID.\v\xFE" CmdOff="" Unit="&lt;v.x&gt;" Analog="false" Text="true" Sensor="true" SourceValHigh="100" DestValHigh="100"/>
	</Comm>
*)
END_ACTION

END_FUNCTION_BLOCK

(* stored: Version 1.1.0.1, ProductVersion 3.1.4024.12
   POU fb_CYDBus6F: Id {b5ad2f58-3dcd-467e-ae4b-ab4e8763d1e5}, SpecialFunc None
   Action ac00_Event: Id {9f48ea95-0266-4afc-8f61-fa8863939c59}
   Action ac01_SetLED: Id {3503c28e-98e0-4224-9478-836ac7f44401}
   Action ac01_SetReset: Id {3250e07b-46b2-446c-b1e6-4aa30407dc3b}
   Action ac01_SetService: Id {94ad80a2-2838-4d36-9fe7-30dfbd3ea1c7}
   Action ac02_Ping: Id {ce16acc0-8d28-4420-a138-108ff038a797}
   Action ac10_Counter: Id {4ce14bda-00cc-4512-9389-ecd907beec5d}
   Action ac99_Doku: Id {b00f08e6-380e-411c-9cf7-802c9da84598} *)
